FUNCTION_BLOCK System_IpcInfo
VAR_INPUT
END_VAR
VAR_OUTPUT
END_VAR
VAR
END_VAR

END_FUNCTION_BLOCK

(* stored: Version 1.1.0.1, ProductVersion 3.1.4024.12
   POU System_IpcInfo: Id {1eda1d9f-cba2-4733-9d4e-4996c44e80f7}, SpecialFunc None *)
